{attribute 'linkalways'} 
{attribute 'no_explicit_call' := 'This FB is a CLASS and must be accessed using methods or properties'}
{attribute 'enable_dynamic_creation'}
FUNCTION_BLOCK _TcVnVector3_USINT EXTENDS AliasDatatypeBase
VAR
	localData : TcVnVector3_USINT;
	activeData : REFERENCE TO TcVnVector3_USINT REF= localData;
	aliasBaseDatatype : _Array0to2OfUSINT;
END_VAR

PROPERTY PUBLIC Address : PVOID
GET
Address := ADR(activeData);
END_GET
END_PROPERTY

METHOD PUBLIC ClearReference
VAR_INPUT
END_VAR
activeData REF= localData;
SetBaseDatatypeReference();
END_METHOD

METHOD PUBLIC Clone : I_Datatype
VAR
    pClone : POINTER TO _TcVnVector3_USINT;
END_VAR
pClone := __NEW(_TcVnVector3_USINT);
Clone := pClone^;
END_METHOD

METHOD FB_init : BOOL
VAR_INPUT
	bInitRetains : BOOL; // if TRUE, the retain variables are initialized (warm start / cold start)
	bInCopyCode : BOOL;  // if TRUE, the instance afterwards gets moved into the copy code (online change)
	//InitialValue : <type>; // if possible, not all values can be initialized
END_VAR
//localData := InitialValue; // if possible, not all values can be initialized
SetBaseDatatypeReference();
AddBaseDatatype(aliasBaseDatatype);
END_METHOD

PROPERTY PUBLIC Identifier : T_MAXSTRING
GET
Identifier := 'TcVnVector3_USINT';
END_GET
END_PROPERTY

METHOD PUBLIC MakeReferenceTo
VAR_INPUT
	ReferenceTarget : REFERENCE TO TcVnVector3_USINT;
END_VAR
activeData REF= ReferenceTarget;
SetBaseDatatypeReference();
END_METHOD

METHOD PROTECTED SetBaseDatatypeReference
VAR_INPUT
END_VAR
aliasBaseDatatype.MakeReferenceTo(activeData);
END_METHOD

PROPERTY PUBLIC Size : UDINT
GET
Size := SIZEOF(activeData);
END_GET
END_PROPERTY

METHOD TryMakeReferenceTo : BOOL
VAR_INPUT
	Target : I_Datatype;
END_VAR
VAR
	targetAsAlias : I_AliasDatatype;
	pTargetData : POINTER TO TcVnVector3_USINT;
END_VAR
IF NOT Target.TryResolveAsAliasDatatype(targetAsAlias) THEN
	RETURN;
END_IF

IF targetAsAlias.Identifier <> Identifier THEN
	RETURN;
END_IF

pTargetData := Target.Address;
activeData REF= pTargetData^;
SetBaseDatatypeReference();
TryMakeReferenceTo := TRUE;
END_METHOD

PROPERTY PUBLIC Value : REFERENCE TO TcVnVector3_USINT
GET
Value REF= activeData;
END_GET
END_PROPERTY

END_FUNCTION_BLOCK

(* stored: Version 1.1.0.1, ProductVersion 3.1.4024.13
   POU _TcVnVector3_USINT: Id {10a4ed3b-923f-0984-2a30-0f52200d2b20}, SpecialFunc None
   Folder Core: Id {e90bb5af-b686-014a-0a80-8e34d52f9c0f}
   Folder Protected: Id {1d485686-62c8-0076-1fde-4138f969088e}
   Folder Customize: Id {27df5931-0334-049a-1dc3-a3478f9d162d}
   Folder Constructor: Id {3e8abd48-370c-0c2d-3a62-9aaac1451386}
   Property Address: Id {bc973d1f-6966-0be2-3310-2823f163b6dd}
   Get Get: Id {93c7ac1b-381e-04a1-333e-b36fcc5f0bda}
   Method ClearReference: Id {57577eee-82ae-03f9-2912-5d6ae0b81756}
   Method Clone: Id {985d1c09-edee-095b-0a10-4ac66ca7a694}
   Method FB_init: Id {0b6682e4-648d-0783-243e-375e5c482fae}
   Property Identifier: Id {19c2bb90-ca93-08e4-3a0a-eb1e6bb6d893}
   Get Get: Id {6567c82a-8008-06af-1f5e-787317389e74}
   Method MakeReferenceTo: Id {7dacde89-e58e-0a5f-2c4a-0fb42aee16bc}
   Method SetBaseDatatypeReference: Id {8c2b08c0-c011-07cc-28a4-010d4b3755a3}
   Property Size: Id {033417f8-fbf5-0fa3-34ad-d280b8bf1186}
   Get Get: Id {c15e7d3f-fa7a-076e-3edd-3798009ff581}
   Method TryMakeReferenceTo: Id {9bf7d28e-734a-08ea-0eca-41710f6476bc}
   Property Value: Id {599d8542-09a3-05e9-1320-a597066fe750}
   Get Get: Id {9dfa7ff1-4a0b-031c-0365-7c6b5e9cab97} *)
